Staubli VAL3: onFunctionSel.pgx

public program onFunctionSel(num x_nIndex, string x_sEvent, num x_nFunctionKey)
  local string l_sMessage
  local string l_sMessage2
  local string l_sSwap
  local num l_nResult
  local bool l_bYes
  local string l_sPath
  local string l_sButton[2]
  local string l_sItem
  local num l_nX
  local num l_nY
  local string l_sString
  local string l_sName
begin
  //
  // do on Key action
  //
  // x_nIndex = actual index item
  // x_sEvent = actual event item
  //
  l_nX=40-use:nBottomX-1
  l_nY=use:nBottomY+1
  switch x_nFunctionKey
    // F1 button
    case 271
    break
    // F2 button
    case 272
    break
    // F3 button
    case 273
      //
      // go to the edit program
      //
      l_sPath=prog:libPath()+"/page_instr"
      l_sItem="HOME1"
      call loadPage(l_sPath,l_sItem)
    break
    // F4 button
    case 274
      //
      // go to the edit program
      //
      l_sPath=prog:libPath()+"/page_instr"
      l_sItem="HOME2"
      call loadPage(l_sPath,l_sItem)
    break
    // F5 button
    case 275
    break
    // F6 button
    case 276
    break
    // F7 button
    case 277
      //
      //
      //
    break
    // F8 button
    case 278
    break
  endSwitch
end
